Staubli VAL3: remSetMode.pgx

program remSetMode(string& sArgs[] (dimensions=1), string& sReturn[] (dimensions=1))
begin
  // Set the remote movement mode to LINEAR or OPTIMAL
  //
  logMsg("call remSetMode")
  if sArgs=="LINEAR"
    bMoveLinear=true
  elseIf sArgs=="OPTIMAL"
    bMoveLinear=false
  else
    call remErrInvalid("SETMODE",sArgs,sReturn)
    return
  endIf
  sReturn="SETMODE "+sArgs
end
